(* IEC 61131-3 sources: trust-platform/examples/communication/ethercat_field_validated_es/src, 2 files *)

(* ---- config.st ---- *)
CONFIGURATION Config
RESOURCE CommEthercatFieldRes ON PLC
    TASK MainTask (INTERVAL := T#10ms, PRIORITY := 1);
    PROGRAM P1 WITH MainTask : Main;
END_RESOURCE
VAR_CONFIG
    P1.DO0 AT %QX0.0 : BOOL;
    P1.DO1 AT %QX0.1 : BOOL;
    P1.DO2 AT %QX0.2 : BOOL;
    P1.DO3 AT %QX0.3 : BOOL;
    P1.DO4 AT %QX0.4 : BOOL;
    P1.DO5 AT %QX0.5 : BOOL;
    P1.DO6 AT %QX0.6 : BOOL;
    P1.DO7 AT %QX0.7 : BOOL;
END_VAR
END_CONFIGURATION

(* ---- main.st ---- *)
PROGRAM Main
VAR
    DO0 : BOOL;
    DO1 : BOOL;
    DO2 : BOOL;
    DO3 : BOOL;
    DO4 : BOOL;
    DO5 : BOOL;
    DO6 : BOOL;
    DO7 : BOOL;

    step_timer : TON;
    step_time : TIME := T#200MS;
    position : INT := 0;
    direction : INT := 1;
END_VAR

step_timer(IN := NOT step_timer.Q, PT := step_time);

IF step_timer.Q THEN
    position := position + direction;
    IF position >= 15 THEN
        direction := -1;
    END_IF;
    IF position <= 0 THEN
        direction := 1;
    END_IF;
END_IF;

IF position <= 7 THEN
    DO0 := (position >= 0);
    DO1 := (position >= 1);
    DO2 := (position >= 2);
    DO3 := (position >= 3);
    DO4 := (position >= 4);
    DO5 := (position >= 5);
    DO6 := (position >= 6);
    DO7 := (position >= 7);
ELSE
    DO0 := (position < 15);
    DO1 := (position < 14);
    DO2 := (position < 13);
    DO3 := (position < 12);
    DO4 := (position < 11);
    DO5 := (position < 10);
    DO6 := (position < 9);
    DO7 := (position < 8);
END_IF;
END_PROGRAM
